PROGRAM PRG_TEST
VAR
	fbRCC_TEST : FB_RCC_TEST;
END_VAR

TcUnit.RUN();

END_PROGRAM

(* stored: Version 1.1.0.1, ProductVersion 3.1.4024.12
   POU PRG_TEST: Id {6ebffb51-15e7-4dae-9c46-bfc01a1da214}, SpecialFunc None *)
